(* Logix 5000 project; controller HP_SSC01hv vendor 1 type 14 code 158 rev 32.11; software revision 32.03; part 11 of 15 *)
(* tags used below, declared in another part *)
   A_S01_0300 : ALIAS FOR System_FaultStandard.0;
   A_S01_0301 : ALIAS FOR System_FaultStandard.1;
   A_S01_0302 : ALIAS FOR System_FaultStandard.2;
   A_S01_0303 : ALIAS FOR System_FaultStandard.3;
   A_S01_0304 : ALIAS FOR System_FaultStandard.4;
   A_S01_0305 : ALIAS FOR System_FaultStandard.5;
   A_S01_0427 : ALIAS FOR System_Warning.27;
   A_S01_0429 : ALIAS FOR System_Warning.29;
   A_S01_0430 : ALIAS FOR System_Warning.30;
   A_S01_0431 : ALIAS FOR System_Warning.31;
   Bit : BOOL;
   C1_ServoStatus : BOOL;
   C1ONS : DINT;
   C2_ServoStatus : BOOL;
   C3_ServoStatus : BOOL;
   Carsl2_Fault_Reset : BOOL;
   Carsl3_Fault_Reset : BOOL;
   DeviceNet_OK : BOOL;
   ErrorMinMaxTotal : REAL[4];
   GroupResetONS : DINT;
   GSV_BSL : CONTROL;
   GSV_BSL_Array : DINT[2];
   GSVTimer : TIMER;
   JoeEnableSERCOScOut : BOOL;
   MasterAtSpeed : BOOL;
   MasterClockCopyMAJ : MOTION_INSTRUCTION;
   MasterClockCopyMAS_Stop1 : MOTION_INSTRUCTION;
   MasterClockCopyMAS_Stop2 : MOTION_INSTRUCTION;
   MasterClockCopyMRP : MOTION_INSTRUCTION;
   MasterClockLocal : AXIS_VIRTUAL;
   MasterClockLocalActualPosition : DINT;
   MasterClockLocalCorrectionAmount : REAL;
   MasterClockTagetTicks : REAL;
   MasterCorrectionStartDelay : TIMER;
   MasterError : REAL;
   MasterErrorCorrectionAtStartONS : BOOL;
   MasterErrorMaxCheck : REAL;
   MasterErrorMinCheck : REAL;
   MasterMinMaxCheck : TIMER;
   MESSAGE_SERCOScOut : MESSAGE;
   Motion : MOTION_GROUP;
   MotionMSGR : MOTION_INSTRUCTION;
   MS_ENBT : DINT[10];
   MS_ENBTRaw : DINT[10];
   none : BOOL;
   NoScan_Comment : BOOL;
   Ons_Fault : DINT;
   ONS_STFault : DINT;
   ProcFaultWord : DINT;
   ProcForceEn : ALIAS FOR ProcForceStatus.1;
   ProcForceExist : ALIAS FOR ProcForceStatus.0;
   ProcForceStatus : DINT;
   ProcLoBattery : ALIAS FOR ProcFaultWord.10;
   ProcRem : BOOL;
   ProcRun : BOOL;
   ProcStatus : DINT;
   Rail_Bypass1 : ALIAS FOR SSC01_Safe1:I.Pt06Data;
   Rail_Bypass2 : ALIAS FOR SSC01_Safe1:I.Pt07Data;
   Rail_Bypass_RIN : REDUNDANT_INPUT;
   RAIL_ENABLE_LH1 : ALIAS FOR SSC01_Safe1:I.Pt00Data;
   RAIL_ENABLE_LH2 : ALIAS FOR SSC01_Safe1:I.Pt01Data;
   RAIL_ENABLE_LH3 : ALIAS FOR SSC01_Safe1:I.Pt02Data;
   RAIL_ENABLE_RH1 : ALIAS FOR SSC01_Safe1:I.Pt03Data;
   RAIL_ENABLE_RH2 : ALIAS FOR SSC01_Safe1:I.Pt04Data;
   RAIL_ENABLE_RH3 : ALIAS FOR SSC01_Safe1:I.Pt05Data;
   RCS_CMD_Auto_TON : TIMER;
   RCS_CMD_BrakeTest : BOOL;
   RCS_CMD_BrakeTest_TON : TIMER;
   RCS_CMD_Evac_TON : TIMER;
   RCS_CMD_EvacToStation : BOOL;
   RCS_CMD_GoNearOnPath : BOOL;
   RCS_CMD_GoNearOnPath_TON : TIMER;
   RCS_Cmd_Mismatch_TON : TIMER;
   RCS_CMD_RunInAuto : BOOL;
   RCS_CMD_Stop1 : BOOL;
   RCS_CMD_Stop2 : BOOL;
   RCS_CMD_Stop_TON : TIMER;
   RCS_Cmd_Unknown : BOOL;
   RCS_MasterClock : ALIAS FOR RCS_SafeMemory_S01.Master_Clock;
   RCS_MasterClockLocalTagetDegrees : REAL;
   RCS_MotionEnable_TON : TIMER;
   RCS_OnPathEnable_TON : TIMER;
   RCS_PwrDisc_AuxA : BOOL;
   RCS_PwrDisc_AuxB : BOOL;
   RCS_PwrDisc_RIN : REDUNDANT_INPUT;
   RCS_PwrDiscA : ALIAS FOR SSC01_Safe2:I.Pt04Data;
   RCS_PwrDiscB : ALIAS FOR SSC01_Safe2:I.Pt05Data;
   RCS_SyncMotionEnable : BOOL;
   RCSMasterGearMAM02 : MOTION_INSTRUCTION;
   S_C1_FaultReset : BOOL;
   S_C2_FaultReset : BOOL;
   S_C3_FaultReset : BOOL;
   S_FaultReset : BOOL;
   S_FlashOff : TIMER;
   S_FlashOn : TIMER;
   S_ONS : BOOL;
   S_RailStateHardware : DINT;
   S_RCS_CMD_FaultReset : BOOL;
   S_RCS_EvacSpeedStart_TON : TIMER;
   S_RCS_MotionCMD_Auto : BOOL;
   S_RCS_MotionCMD_BrakeTest : BOOL;
   S_RCS_MotionCMD_Evac : BOOL;
   S_RCS_MotionCMD_GoNearOnPath : BOOL;
   S_RCS_MotionCMD_Stop1 : BOOL;
   S_RCS_MotionCMD_Stop2 : BOOL;
   S_RCS_MotionEnable : BOOL;
   S_RCS_RailStateEthernet : ALIAS FOR RCS_SafeMemory_S01.RailStateEthernet;
   S_RCS_RailStateHardwareUnknown : DINT;
   S_SSC_InputsOK : BOOL;
   SafetySignatureGSVTimer : TIMER;
   SafetySignatureSINT : SINT[50];
   SafetySignatureString : STRING;
   SSC_Rail_BypassOK : BOOL;
   ST_NoScan_Comment : BOOL;
   STS_Enable_Rail : DINT;
   STS_Rail_Bypass_InputOK : BOOL;
   STS_RCS_PwrDisc_InputOK : BOOL;
   STS_SSC_Safety_NodesOK : BOOL;
   STS_Status_OK : BOOL;
   System_FaultStandard : DINT;
   System_Warning : DINT;
   Tmr_Rail_Bypass_Disc : TIMER;
   Tmr_Rail_Debn : TIMER;

PROGRAM Main_SSC   (* main routine M00_Main *)

ROUTINE M00_Main   (* ladder *)
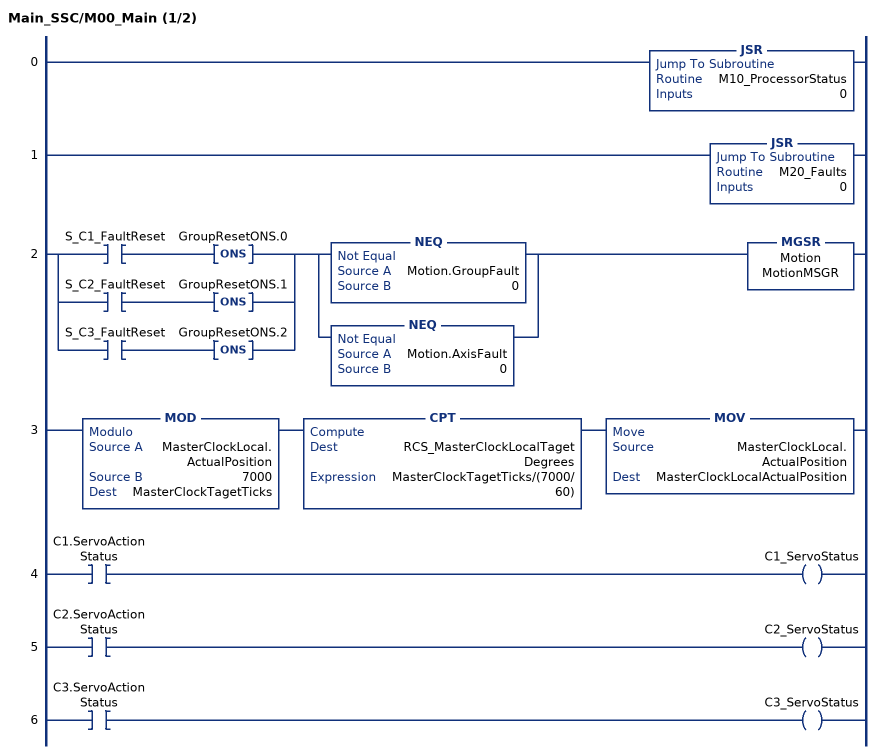
   0: JSR(M10_ProcessorStatus,0);
   1: JSR(M20_Faults,0);
   2: [XIC(S_C1_FaultReset) ONS(GroupResetONS.0) ,XIC(S_C2_FaultReset) ONS(GroupResetONS.1) ,XIC(S_C3_FaultReset) ONS(GroupResetONS.2) ][NEQ(Motion.GroupFault,0) ,NEQ(Motion.AxisFault,0) ]MGSR(Motion,MotionMSGR);
   3: MOD(MasterClockLocal.ActualPosition,7000,MasterClockTagetTicks)CPT(RCS_MasterClockLocalTagetDegrees,MasterClockTagetTicks/(7000/60))MOV(MasterClockLocal.ActualPosition,MasterClockLocalActualPosition);
   4: XIC(C1.ServoActionStatus)OTE(C1_ServoStatus);
   5: XIC(C2.ServoActionStatus)OTE(C2_ServoStatus);
   6: XIC(C3.ServoActionStatus)OTE(C3_ServoStatus);
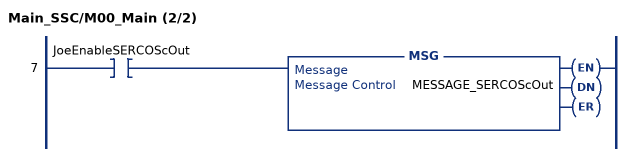
   7: XIC(JoeEnableSERCOScOut)MSG(MESSAGE_SERCOScOut);
END_ROUTINE

ROUTINE M10_ProcessorStatus   (* ladder *)
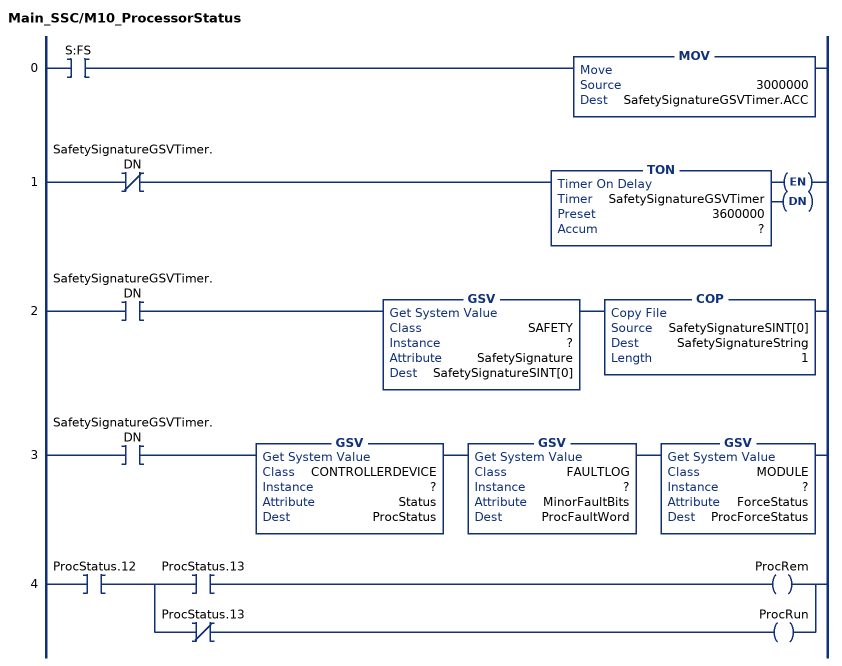
   0: XIC(S:FS)MOV(3000000,SafetySignatureGSVTimer.ACC);
   1: XIO(SafetySignatureGSVTimer.DN)TON(SafetySignatureGSVTimer,?,?);
   2: XIC(SafetySignatureGSVTimer.DN)GSV(SAFETY,?,SafetySignature,SafetySignatureSINT[0])COP(SafetySignatureSINT[0],SafetySignatureString,1);
   3: XIC(SafetySignatureGSVTimer.DN)GSV(CONTROLLERDEVICE,?,Status,ProcStatus)GSV(FAULTLOG,?,MinorFaultBits,ProcFaultWord)GSV(MODULE,?,ForceStatus,ProcForceStatus);
   4: XIC(ProcStatus.12)[XIC(ProcStatus.13) OTE(ProcRem) ,XIO(ProcStatus.13) OTE(ProcRun) ];
END_ROUTINE

ROUTINE M20_Faults   (* ladder *)
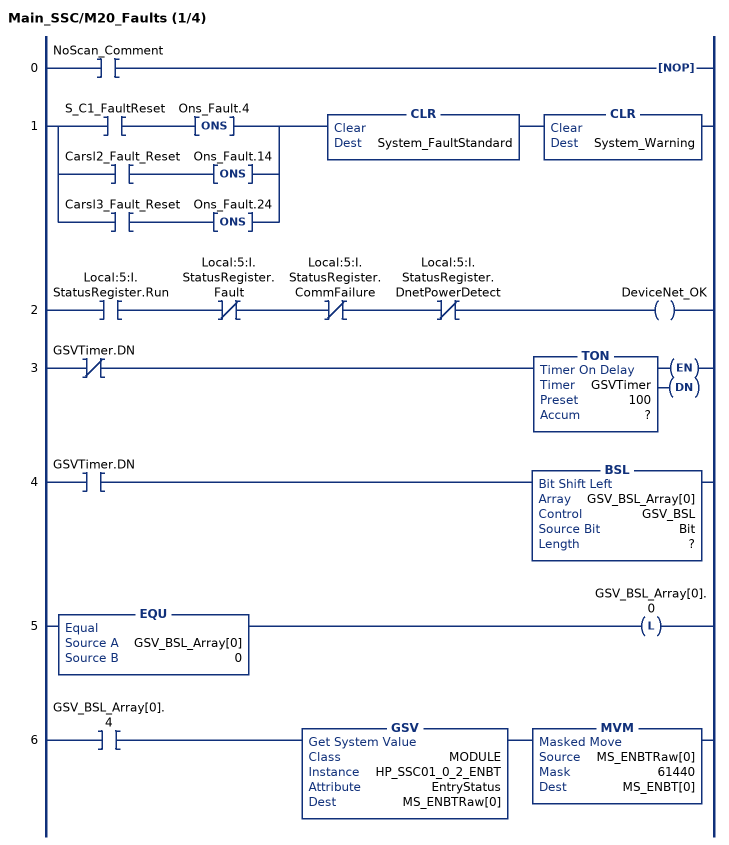
   0: XIC(NoScan_Comment)NOP();
   1: [XIC(S_C1_FaultReset) ONS(Ons_Fault.4) ,XIC(Carsl2_Fault_Reset) ONS(Ons_Fault.14) ,XIC(Carsl3_Fault_Reset) ONS(Ons_Fault.24) ]CLR(System_FaultStandard)CLR(System_Warning);
   2: XIC(Local:5:I.StatusRegister.Run)XIO(Local:5:I.StatusRegister.Fault)XIO(Local:5:I.StatusRegister.CommFailure)XIO(Local:5:I.StatusRegister.DnetPowerDetect)OTE(DeviceNet_OK);
   3: XIO(GSVTimer.DN)TON(GSVTimer,?,?);
   4: XIC(GSVTimer.DN)BSL(GSV_BSL_Array[0],GSV_BSL,Bit,?);
   5: EQU(GSV_BSL_Array[0],0)OTL(GSV_BSL_Array[0].0);
   6: XIC(GSV_BSL_Array[0].4)GSV(MODULE,HP_SSC01_0_2_ENBT,EntryStatus,MS_ENBTRaw[0])MVM(MS_ENBTRaw[0],61440,MS_ENBT[0]);
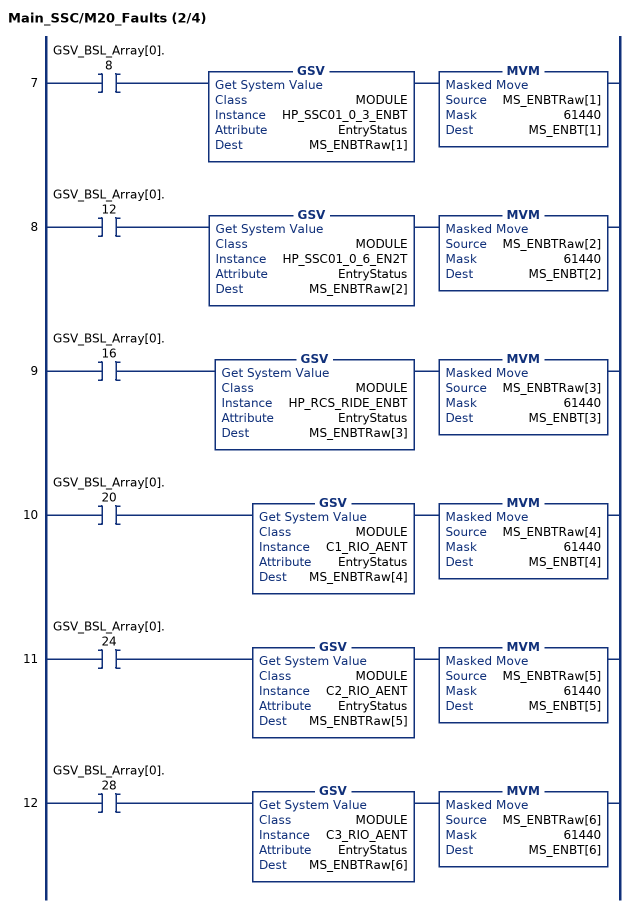
   7: XIC(GSV_BSL_Array[0].8)GSV(MODULE,HP_SSC01_0_3_ENBT,EntryStatus,MS_ENBTRaw[1])MVM(MS_ENBTRaw[1],61440,MS_ENBT[1]);
   8: XIC(GSV_BSL_Array[0].12)GSV(MODULE,HP_SSC01_0_6_EN2T,EntryStatus,MS_ENBTRaw[2])MVM(MS_ENBTRaw[2],61440,MS_ENBT[2]);
   9: XIC(GSV_BSL_Array[0].16)GSV(MODULE,HP_RCS_RIDE_ENBT,EntryStatus,MS_ENBTRaw[3])MVM(MS_ENBTRaw[3],61440,MS_ENBT[3]);
   10: XIC(GSV_BSL_Array[0].20)GSV(MODULE,C1_RIO_AENT,EntryStatus,MS_ENBTRaw[4])MVM(MS_ENBTRaw[4],61440,MS_ENBT[4]);
   11: XIC(GSV_BSL_Array[0].24)GSV(MODULE,C2_RIO_AENT,EntryStatus,MS_ENBTRaw[5])MVM(MS_ENBTRaw[5],61440,MS_ENBT[5]);
   12: XIC(GSV_BSL_Array[0].28)GSV(MODULE,C3_RIO_AENT,EntryStatus,MS_ENBTRaw[6])MVM(MS_ENBTRaw[6],61440,MS_ENBT[6]);
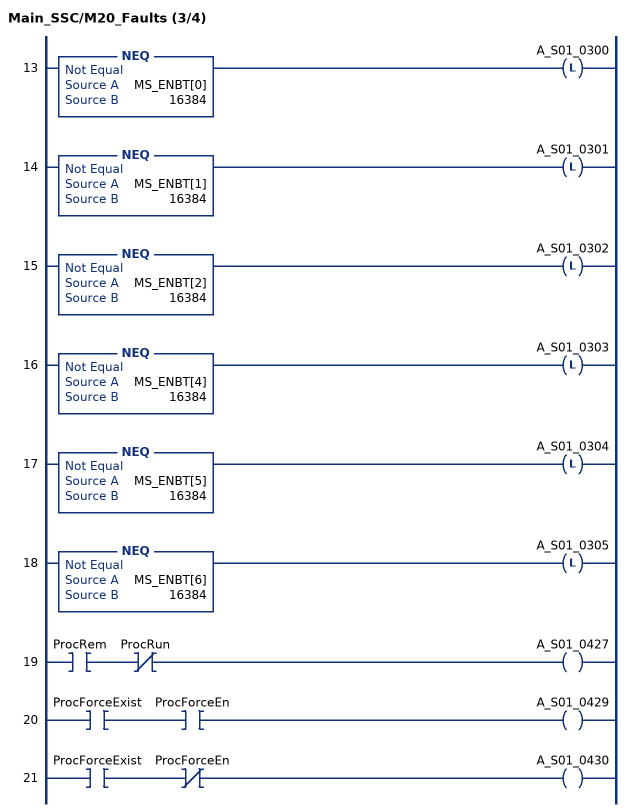
   13: NEQ(MS_ENBT[0],16384)OTL(A_S01_0300);
   14: NEQ(MS_ENBT[1],16384)OTL(A_S01_0301);
   15: NEQ(MS_ENBT[2],16384)OTL(A_S01_0302);
   16: NEQ(MS_ENBT[4],16384)OTL(A_S01_0303);
   17: NEQ(MS_ENBT[5],16384)OTL(A_S01_0304);
   18: NEQ(MS_ENBT[6],16384)OTL(A_S01_0305);
   19: XIC(ProcRem)XIO(ProcRun)OTE(A_S01_0427);
   20: XIC(ProcForceExist)XIC(ProcForceEn)OTE(A_S01_0429);
   21: XIC(ProcForceExist)XIO(ProcForceEn)OTE(A_S01_0430);
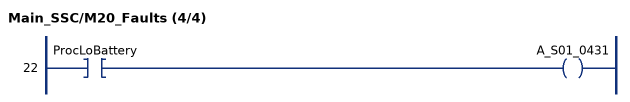
   22: XIC(ProcLoBattery)OTE(A_S01_0431);
END_ROUTINE
END_PROGRAM

PROGRAM MasterCopy   (* main routine C400_Main *)

ROUTINE C400_Main   (* ladder *)
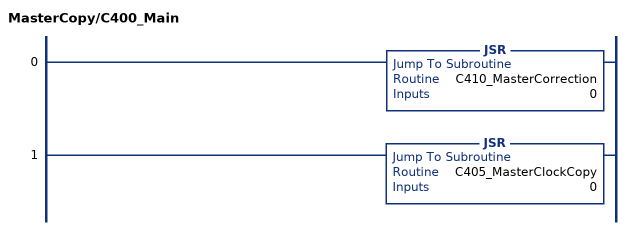
   0: JSR(C410_MasterCorrection,0);
   1: JSR(C405_MasterClockCopy,0);
END_ROUTINE

ROUTINE C405_MasterClockCopy   (* ladder *)
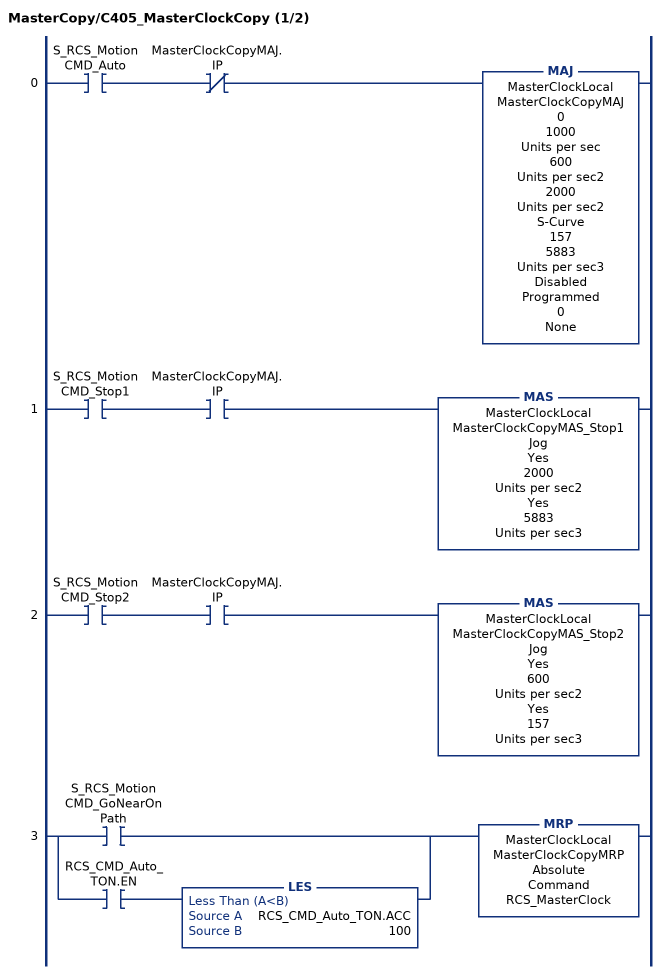
   0: XIC(S_RCS_MotionCMD_Auto)XIO(MasterClockCopyMAJ.IP)MAJ(MasterClockLocal,MasterClockCopyMAJ,0,1000,Units per sec,600,Units per sec2,2000,Units per sec2,S-Curve,157,5883,Units per sec3,Disabled,Programmed,0,None);
   1: XIC(S_RCS_MotionCMD_Stop1)XIC(MasterClockCopyMAJ.IP)MAS(MasterClockLocal,MasterClockCopyMAS_Stop1,Jog,Yes,2000,Units per sec2,Yes,5883,Units per sec3);
   2: XIC(S_RCS_MotionCMD_Stop2)XIC(MasterClockCopyMAJ.IP)MAS(MasterClockLocal,MasterClockCopyMAS_Stop2,Jog,Yes,600,Units per sec2,Yes,157,Units per sec3);
   3: [XIC(S_RCS_MotionCMD_GoNearOnPath) ,XIC(RCS_CMD_Auto_TON.EN) LES(RCS_CMD_Auto_TON.ACC,100) ]MRP(MasterClockLocal,MasterClockCopyMRP,Absolute,Command,RCS_MasterClock);
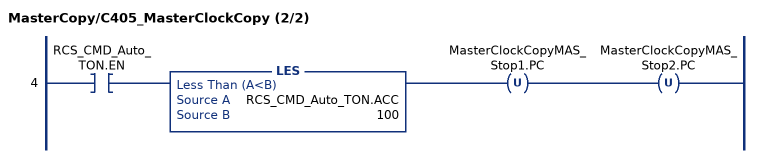
   4: XIC(RCS_CMD_Auto_TON.EN)LES(RCS_CMD_Auto_TON.ACC,100)OTU(MasterClockCopyMAS_Stop1.PC)OTU(MasterClockCopyMAS_Stop2.PC);
END_ROUTINE

ROUTINE C410_MasterCorrection   (* ladder *)
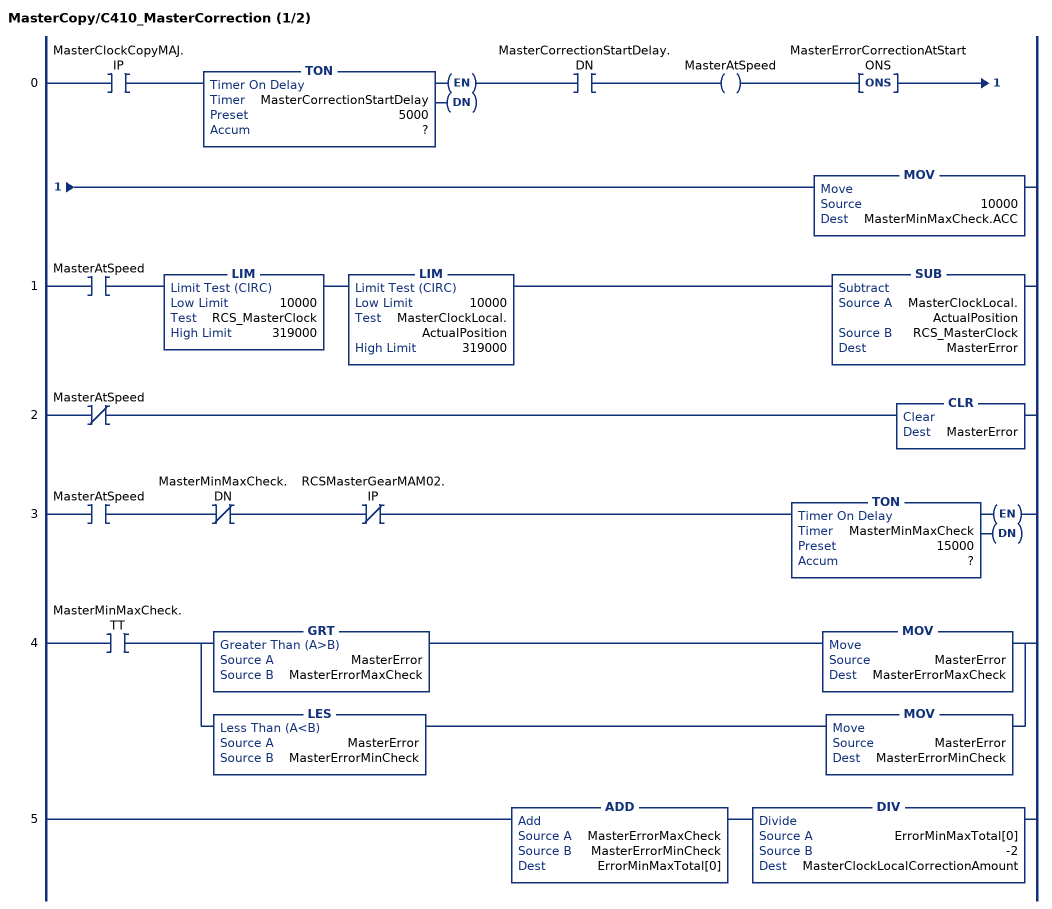
   0: XIC(MasterClockCopyMAJ.IP)TON(MasterCorrectionStartDelay,?,?)XIC(MasterCorrectionStartDelay.DN)OTE(MasterAtSpeed)ONS(MasterErrorCorrectionAtStartONS)MOV(10000,MasterMinMaxCheck.ACC);
   1: XIC(MasterAtSpeed)LIM(10000,RCS_MasterClock,319000)LIM(10000,MasterClockLocal.ActualPosition,319000)SUB(MasterClockLocal.ActualPosition,RCS_MasterClock,MasterError);
   2: XIO(MasterAtSpeed)CLR(MasterError);
   3: XIC(MasterAtSpeed)XIO(MasterMinMaxCheck.DN)XIO(RCSMasterGearMAM02.IP)TON(MasterMinMaxCheck,?,?);
   4: XIC(MasterMinMaxCheck.TT)[GRT(MasterError,MasterErrorMaxCheck) MOV(MasterError,MasterErrorMaxCheck) ,LES(MasterError,MasterErrorMinCheck) MOV(MasterError,MasterErrorMinCheck) ];
   5: ADD(MasterErrorMaxCheck,MasterErrorMinCheck,ErrorMinMaxTotal[0])DIV(ErrorMinMaxTotal[0],-2,MasterClockLocalCorrectionAmount);
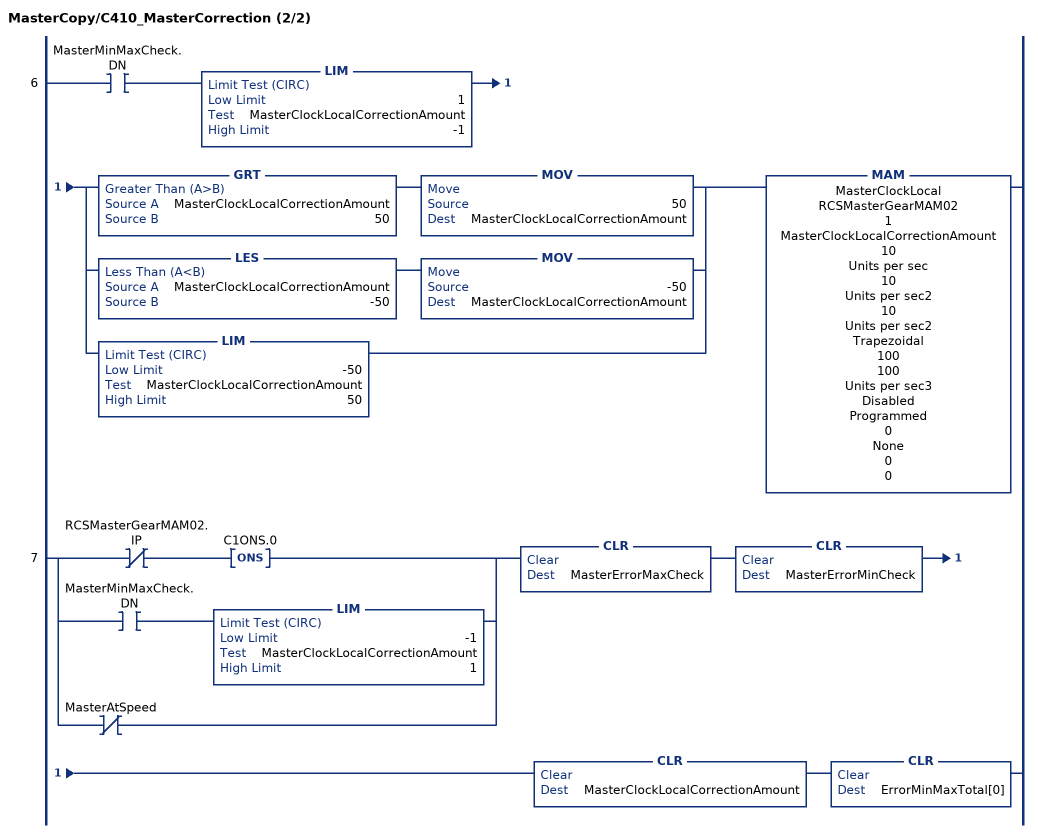
   6: XIC(MasterMinMaxCheck.DN)LIM(1,MasterClockLocalCorrectionAmount,-1)[GRT(MasterClockLocalCorrectionAmount,50) MOV(50,MasterClockLocalCorrectionAmount) ,LES(MasterClockLocalCorrectionAmount,-50) MOV(-50,MasterClockLocalCorrectionAmount) ,LIM(-50,MasterClockLocalCorrectionAmount,50) ]MAM(MasterClockLocal,RCSMasterGearMAM02,1,MasterClockLocalCorrectionAmount,10,Units per sec,10,Units per sec2,10,Units per sec2,Trapezoidal,100,100,Units per sec3,Disabled,Programmed,0,None,0,0);
   7: [XIO(RCSMasterGearMAM02.IP) ONS(C1ONS.0) ,XIC(MasterMinMaxCheck.DN) LIM(-1,MasterClockLocalCorrectionAmount,1) ,XIO(MasterAtSpeed) ]CLR(MasterErrorMaxCheck)CLR(MasterErrorMinCheck)CLR(MasterClockLocalCorrectionAmount)CLR(ErrorMinMaxTotal[0]);
END_ROUTINE
END_PROGRAM

PROGRAM Safe_SSC   (* main routine ST00_Main, safety *)

ROUTINE ST00_Main   (* ladder *)
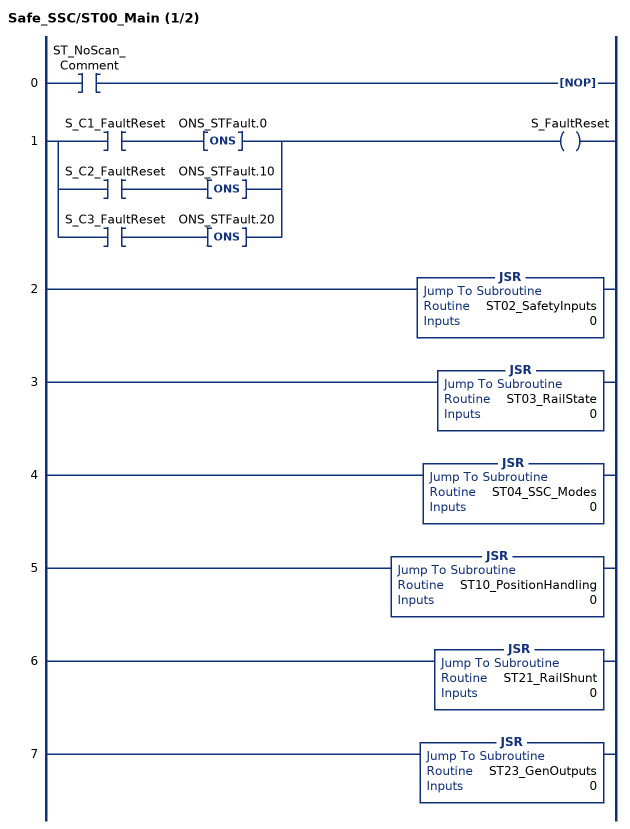
   0: XIC(ST_NoScan_Comment)NOP();
   1: [XIC(S_C1_FaultReset) ONS(ONS_STFault.0) ,XIC(S_C2_FaultReset) ONS(ONS_STFault.10) ,XIC(S_C3_FaultReset) ONS(ONS_STFault.20) ]OTE(S_FaultReset);
   2: JSR(ST02_SafetyInputs,0);
   3: JSR(ST03_RailState,0);
   4: JSR(ST04_SSC_Modes,0);
   5: JSR(ST10_PositionHandling,0);
   6: JSR(ST21_RailShunt,0);
   7: JSR(ST23_GenOutputs,0);
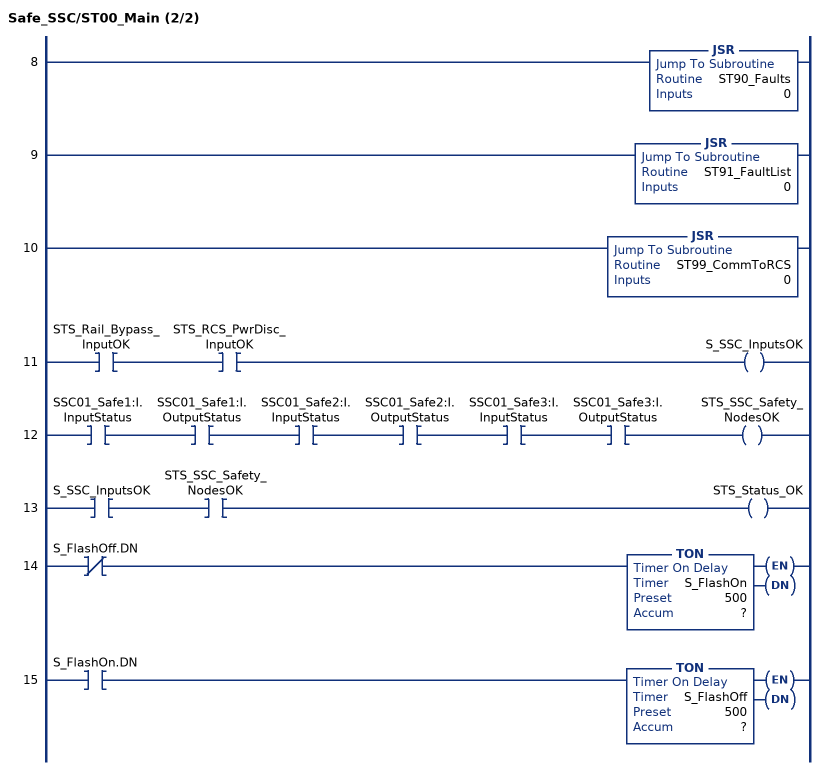
   8: JSR(ST90_Faults,0);
   9: JSR(ST91_FaultList,0);
   10: JSR(ST99_CommToRCS,0);
   11: XIC(STS_Rail_Bypass_InputOK)XIC(STS_RCS_PwrDisc_InputOK)OTE(S_SSC_InputsOK);
   12: XIC(SSC01_Safe1:I.InputStatus)XIC(SSC01_Safe1:I.OutputStatus)XIC(SSC01_Safe2:I.InputStatus)XIC(SSC01_Safe2:I.OutputStatus)XIC(SSC01_Safe3:I.InputStatus)XIC(SSC01_Safe3:I.OutputStatus)OTE(STS_SSC_Safety_NodesOK);
   13: XIC(S_SSC_InputsOK)XIC(STS_SSC_Safety_NodesOK)OTE(STS_Status_OK);
   14: XIO(S_FlashOff.DN)TON(S_FlashOn,?,?);
   15: XIC(S_FlashOn.DN)TON(S_FlashOff,?,?);
END_ROUTINE

ROUTINE ST02_SafetyInputs   (* ladder *)
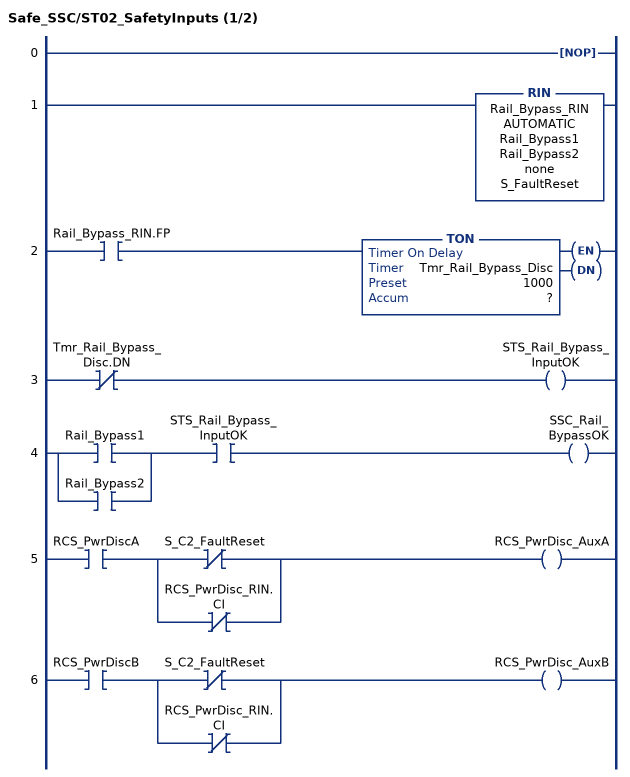
   0: NOP();
   1: RIN(Rail_Bypass_RIN,AUTOMATIC,Rail_Bypass1,Rail_Bypass2,none,S_FaultReset);
   2: XIC(Rail_Bypass_RIN.FP)TON(Tmr_Rail_Bypass_Disc,?,?);
   3: XIO(Tmr_Rail_Bypass_Disc.DN)OTE(STS_Rail_Bypass_InputOK);
   4: [XIC(Rail_Bypass1) ,XIC(Rail_Bypass2) ]XIC(STS_Rail_Bypass_InputOK)OTE(SSC_Rail_BypassOK);
   5: XIC(RCS_PwrDiscA)[XIO(S_C2_FaultReset) ,XIO(RCS_PwrDisc_RIN.CI) ]OTE(RCS_PwrDisc_AuxA);
   6: XIC(RCS_PwrDiscB)[XIO(S_C2_FaultReset) ,XIO(RCS_PwrDisc_RIN.CI) ]OTE(RCS_PwrDisc_AuxB);
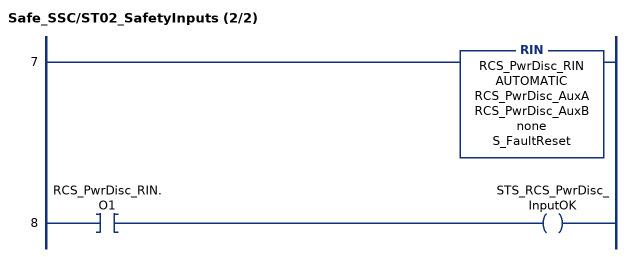
   7: RIN(RCS_PwrDisc_RIN,AUTOMATIC,RCS_PwrDisc_AuxA,RCS_PwrDisc_AuxB,none,S_FaultReset);
   8: XIC(RCS_PwrDisc_RIN.O1)OTE(STS_RCS_PwrDisc_InputOK);
END_ROUTINE

ROUTINE ST03_RailState   (* ladder *)
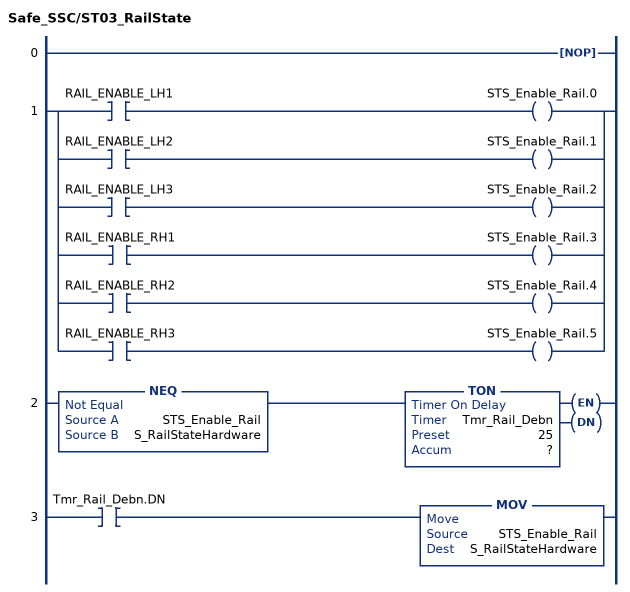
   0: NOP();
   1: [XIC(RAIL_ENABLE_LH1) OTE(STS_Enable_Rail.0) ,XIC(RAIL_ENABLE_LH2) OTE(STS_Enable_Rail.1) ,XIC(RAIL_ENABLE_LH3) OTE(STS_Enable_Rail.2) ,XIC(RAIL_ENABLE_RH1) OTE(STS_Enable_Rail.3) ,XIC(RAIL_ENABLE_RH2) OTE(STS_Enable_Rail.4) ,XIC(RAIL_ENABLE_RH3) OTE(STS_Enable_Rail.5) ];
   2: NEQ(STS_Enable_Rail,S_RailStateHardware)TON(Tmr_Rail_Debn,?,?);
   3: XIC(Tmr_Rail_Debn.DN)MOV(STS_Enable_Rail,S_RailStateHardware);
END_ROUTINE

ROUTINE ST04_SSC_Modes   (* ladder *)
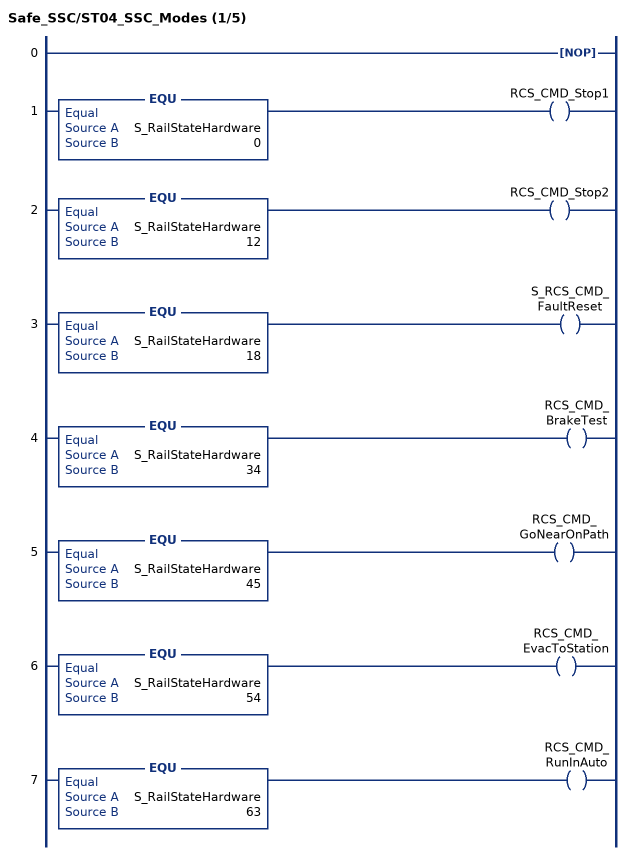
   0: NOP();
   1: EQU(S_RailStateHardware,0)OTE(RCS_CMD_Stop1);
   2: EQU(S_RailStateHardware,12)OTE(RCS_CMD_Stop2);
   3: EQU(S_RailStateHardware,18)OTE(S_RCS_CMD_FaultReset);
   4: EQU(S_RailStateHardware,34)OTE(RCS_CMD_BrakeTest);
   5: EQU(S_RailStateHardware,45)OTE(RCS_CMD_GoNearOnPath);
   6: EQU(S_RailStateHardware,54)OTE(RCS_CMD_EvacToStation);
   7: EQU(S_RailStateHardware,63)OTE(RCS_CMD_RunInAuto);
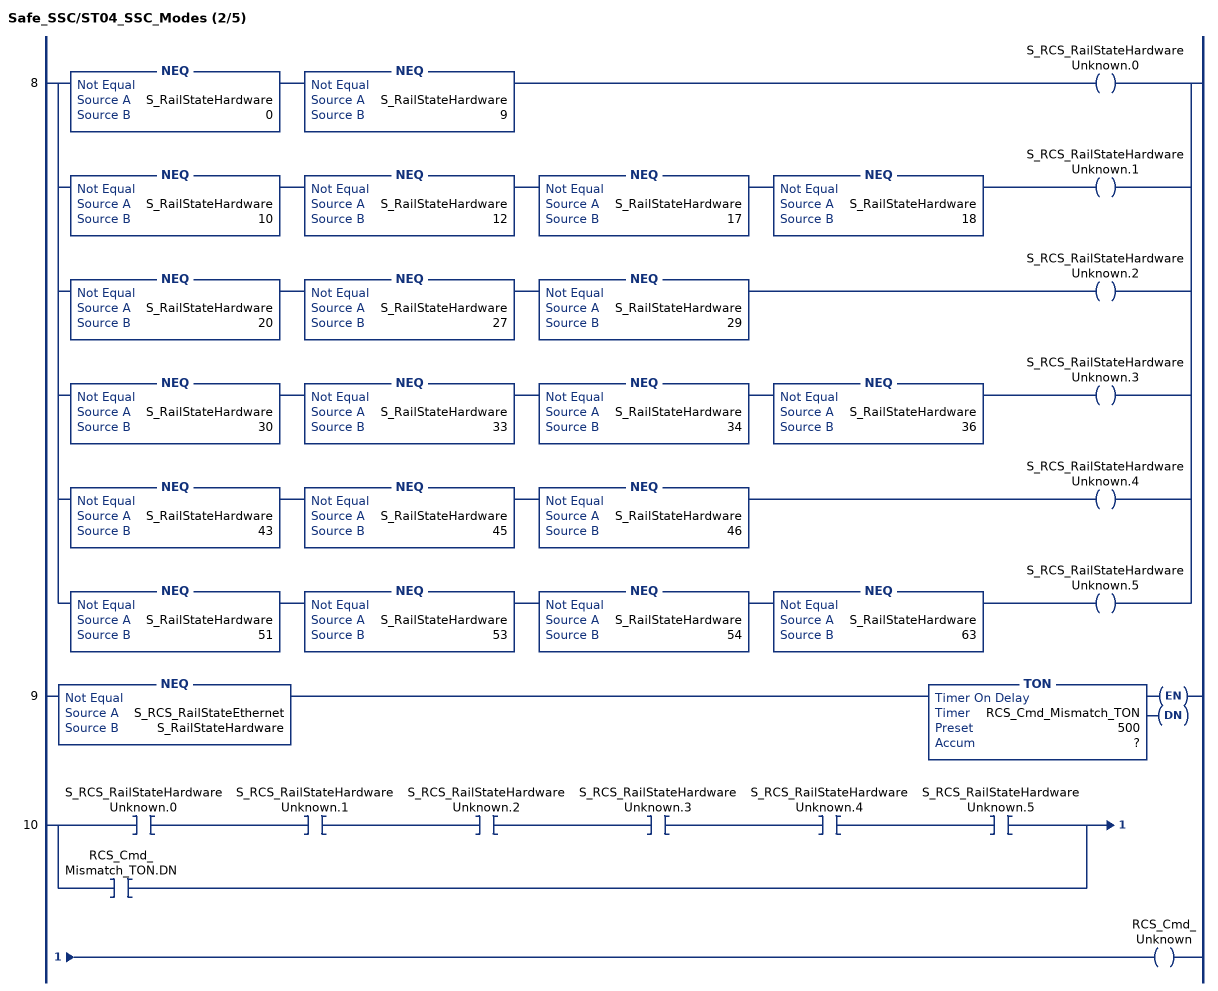
   8: [NEQ(S_RailStateHardware,0) NEQ(S_RailStateHardware,9) OTE(S_RCS_RailStateHardwareUnknown.0) ,NEQ(S_RailStateHardware,10) NEQ(S_RailStateHardware,12) NEQ(S_RailStateHardware,17) NEQ(S_RailStateHardware,18) OTE(S_RCS_RailStateHardwareUnknown.1) ,NEQ(S_RailStateHardware,20) NEQ(S_RailStateHardware,27) NEQ(S_RailStateHardware,29) OTE(S_RCS_RailStateHardwareUnknown.2) ,NEQ(S_RailStateHardware,30) NEQ(S_RailStateHardware,33) NEQ(S_RailStateHardware,34) NEQ(S_RailStateHardware,36) OTE(S_RCS_RailStateHardwareUnknown.3) ,NEQ(S_RailStateHardware,43) NEQ(S_RailStateHardware,45) NEQ(S_RailStateHardware,46) OTE(S_RCS_RailStateHardwareUnknown.4) ,NEQ(S_RailStateHardware,51) NEQ(S_RailStateHardware,53) NEQ(S_RailStateHardware,54) NEQ(S_RailStateHardware,63) OTE(S_RCS_RailStateHardwareUnknown.5) ];
   9: NEQ(S_RCS_RailStateEthernet,S_RailStateHardware)TON(RCS_Cmd_Mismatch_TON,?,?);
   10: [XIC(S_RCS_RailStateHardwareUnknown.0) XIC(S_RCS_RailStateHardwareUnknown.1) XIC(S_RCS_RailStateHardwareUnknown.2) XIC(S_RCS_RailStateHardwareUnknown.3) XIC(S_RCS_RailStateHardwareUnknown.4) XIC(S_RCS_RailStateHardwareUnknown.5) ,XIC(RCS_Cmd_Mismatch_TON.DN) ]OTE(RCS_Cmd_Unknown);
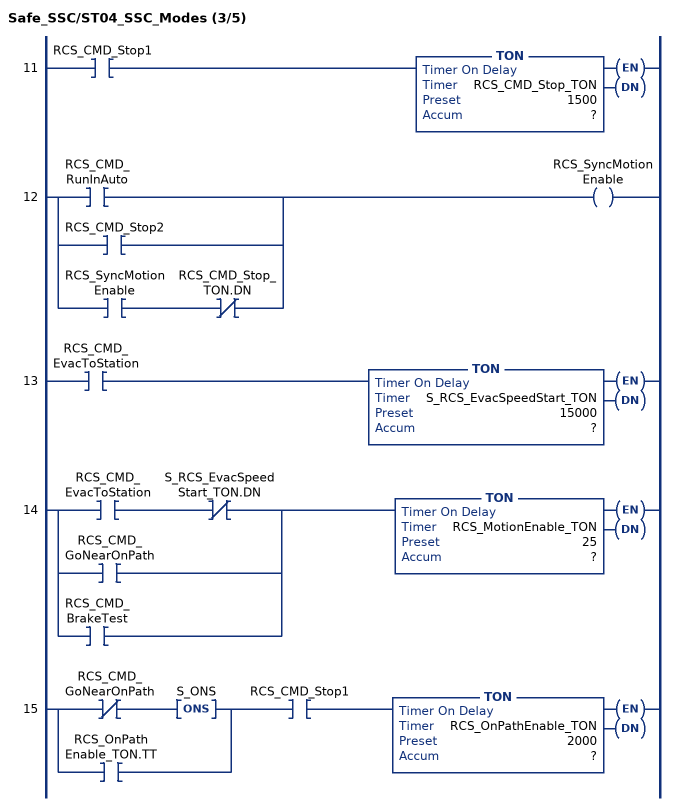
   11: XIC(RCS_CMD_Stop1)TON(RCS_CMD_Stop_TON,?,?);
   12: [XIC(RCS_CMD_RunInAuto) ,XIC(RCS_CMD_Stop2) ,XIC(RCS_SyncMotionEnable) XIO(RCS_CMD_Stop_TON.DN) ]OTE(RCS_SyncMotionEnable);
   13: XIC(RCS_CMD_EvacToStation)TON(S_RCS_EvacSpeedStart_TON,?,?);
   14: [XIC(RCS_CMD_EvacToStation) XIO(S_RCS_EvacSpeedStart_TON.DN) ,XIC(RCS_CMD_GoNearOnPath) ,XIC(RCS_CMD_BrakeTest) ]TON(RCS_MotionEnable_TON,?,?);
   15: [XIO(RCS_CMD_GoNearOnPath) ONS(S_ONS) ,XIC(RCS_OnPathEnable_TON.TT) ]XIC(RCS_CMD_Stop1)TON(RCS_OnPathEnable_TON,?,?);
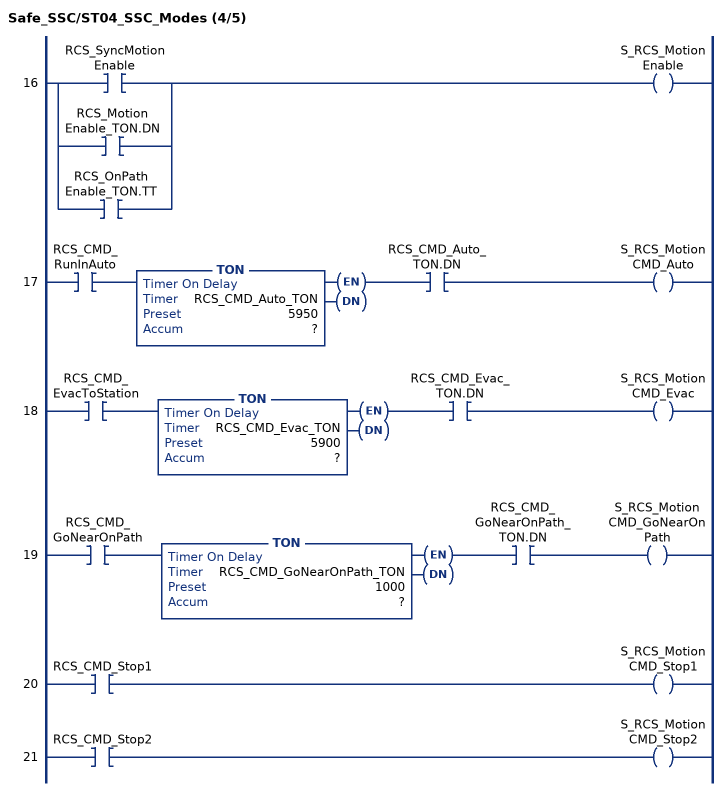
   16: [XIC(RCS_SyncMotionEnable) ,XIC(RCS_MotionEnable_TON.DN) ,XIC(RCS_OnPathEnable_TON.TT) ]OTE(S_RCS_MotionEnable);
   17: XIC(RCS_CMD_RunInAuto)TON(RCS_CMD_Auto_TON,?,?)XIC(RCS_CMD_Auto_TON.DN)OTE(S_RCS_MotionCMD_Auto);
   18: XIC(RCS_CMD_EvacToStation)TON(RCS_CMD_Evac_TON,?,?)XIC(RCS_CMD_Evac_TON.DN)OTE(S_RCS_MotionCMD_Evac);
   19: XIC(RCS_CMD_GoNearOnPath)TON(RCS_CMD_GoNearOnPath_TON,?,?)XIC(RCS_CMD_GoNearOnPath_TON.DN)OTE(S_RCS_MotionCMD_GoNearOnPath);
   20: XIC(RCS_CMD_Stop1)OTE(S_RCS_MotionCMD_Stop1);
   21: XIC(RCS_CMD_Stop2)OTE(S_RCS_MotionCMD_Stop2);
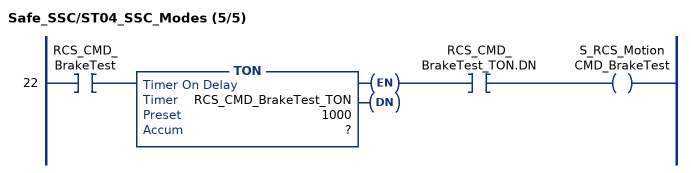
   22: XIC(RCS_CMD_BrakeTest)TON(RCS_CMD_BrakeTest_TON,?,?)XIC(RCS_CMD_BrakeTest_TON.DN)OTE(S_RCS_MotionCMD_BrakeTest);
END_ROUTINE
